// TIA Portal V17 export
// export: Created 2026-04-13T11:12:44.1756721Z, ExportSetting WithDefaults, DisplayName Totally Integrated Automation Portal, DisplayVersion V17 Update 4, DisplayName TIA Portal Openness, DisplayVersion V17 Update 4, DisplayName TIA Portal Version Control Interface, DisplayVersion V17, DisplayName SINAMICS Startdrive Advanced, DisplayVersion V17, DisplayName SINAMICS Startdrive G130, G150, S120, S150, SINAMICS MV, S210, DisplayVersion V17, DisplayName SINAMICS Startdrive G110M, G120, G120C, G120D, G120P, G115D, DisplayVersion V17, DisplayName STEP 7 Professional, DisplayVersion V17 Update 4, DisplayName STEP 7 Safety, DisplayVersion V17, DisplayName WinCC Professional, DisplayVersion V17 Update 4
FUNCTION_BLOCK "12-2点斜率输入->输出"   // FB41, LAD
{ S7_Optimized_Access := 'TRUE' }
VERSION : 0.1
// stored: AutoNumber true, IsIECCheckEnabled false, IsRetainMemResEnabled false, MemoryReserve 100, SetENOAutomatically false, UDAEnableTagReadback false
   VAR_INPUT
      sr输入ok : Real;
   END_VAR
   VAR_OUTPUT
      sc输出ok : Int;
   END_VAR
   VAR_IN_OUT
      sr输入1 : Real;
      sc输出1 : Real;
      sr输入2 : Real;
      sc输出2 : Real;
   END_VAR
BEGIN

REGION Network 1 (SCL)


   #sc输出ok := REAL_TO_INT(((#sc输出2 - #sc输出1) / (#sr输入2 - #sr输入1)) * #sr输入ok);
END_REGION
END_FUNCTION_BLOCK
